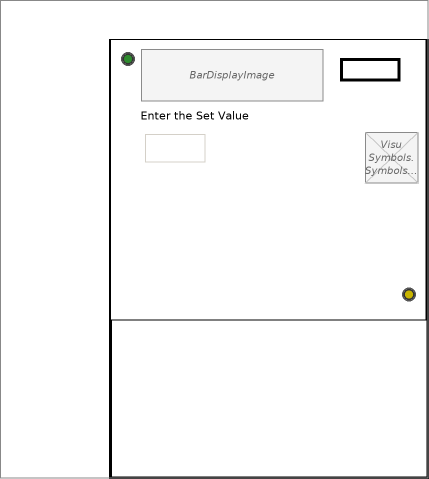
VISUALIZATION Visualization  // 429x479
    Rectangle (109,39 320x440)
    Rectangle (110,39 316x281)
    RoundedRectangle (340,58 60x23), tooltip "Handle to open Fridge Door"
        OnMouseClick: toggle GVL_Var.bDoorOpen
    Image (365,132 53x51), angle 182, tooltip "Fridge Lamp which light the Interior", invisible if: NOT GVL_Var.bLamp, image: VisuSymbols.Symbols.light
        p2175578022: GVL_Var.bLamp
    Textfield (145,134 60x28), tooltip "Set the Temp to be maintained in Fridge between 0 and 20", text variable: GVL_Var.fTempSet
        OnMouseClick: write the text variable via Default, min 0, max 20
    Lamp1 (401,283 16x23), tooltip "Indicates when Fridge Door opened for long time", variable: GVL_Var.bSignal, style: Lamp-Lamp1-Yellow
    Lamp1 (120,49 16x20), tooltip "State of Compressor", variable: GVL_Var.bCompressor, style: Lamp-Lamp1-Green
    BarDisplayImage (141,49 182x52), value: GVL_Var.fTempActual, style: BarDisplayImage-Gray, scale format: %.1f, scale 0..20
    Label (120,101 150x30), "Enter the Set Value"
END_VISUALIZATION

(* stored: Version 1.1.0.1, ProductVersion 3.1.4024.4
   Visu Visualization: Id {0dbe2b12-4493-4860-b7e6-523b6b3df4d3} *)
